(* Logix 5000 project; controller QW361 vendor 1 type 14 code 107 rev 32.11; software revision 32.00; part 20 of 20 *)
(* tags used below, declared in another part *)
   DG1 : MOTOR;   // Diesel generator
   FIT001 : PRANALOG;   // Station discharge flow
   FIT001_CA : ALM;   // Station discharge flow calibrate mode alarm
   FIT001_FL : ALM;   // Station discharge flow sensor fail alarm
   FIT001_hh : ALM;   // Station discharge flow high high alarm
   FIT001_hi : ALM;   // Station discharge flow high alarm
   FIT001_ll : ALM;   // Station discharge flow low low alarm
   FIT001_lo : ALM;   // Station discharge flow low alarm
   FunctionBlock_Cycle_Time : REAL;   // Main Task Cycle Time in mseconds
   LIT001 : PRANALOG;   // Wet well level
   LIT001_CA : ALM;   // Wet well level calibrate mode alarm
   LIT001_FL : ALM;   // Wet well level sensor fail alarm
   LIT001_hh : ALM;   // Wet well level high high alarm
   LIT001_hi : ALM;   // Wet well level high alarm
   LIT001_ll : ALM;   // Wet well level low low alarm
   LIT001_lo : ALM;   // Wet well level low alarm
   P001 : MOTOR;   // Raw sewage pump 1
   P002 : MOTOR;   // Raw sewage pump 2
   pranalog_pwrup_done : BOOL;
   report15_data : LogRecord15[800];
   report15_row_qty : DINT;
   report5_data : LogRecord5[2400];
   report5_row_qty : DINT;
   report_data : LogRecord[200];
   report_pwrup_done : BOOL;
   report_row_qty : DINT;
   sequence_pwrup_done : BOOL;
   valve_pwrup_done : BOOL;
   WALLCLOCK : DateTime;   // Global date / time
   WALLCLOCK_lock : BOOL;

PROGRAM PranalogProgram   (* main routine Pranalogs *)
VAR
   pranalog : PRANALOG := (MaxEU := 20.0, raw := -0.00625, valid := 1, log := 1, hihiraw := 1, hiraw := 1);
   ratio : REAL;
END_VAR

ROUTINE PranalogRoutine   (* structured text *)
   SBR(pranalog);
   
   (* Pranalog function block *)
   
   (* Does all processing for process analogs *)
   
   (* Calling parameters: *)
   (*     pranalog : PRANALOG *)
   
   (* Globals used: *)
   (*     functionblocktask_cycle_time *)
   
   (* Globals changed: *)
   
   (*-------------------------------------------------------------------------------------------------------------------------------------------------*)
   
   
   (* handle the processed analogs *)
   
   (* if not in calibrate mode and not hold and pranalog.calc is not NAN, set the output to calc, smoothed by lag *)
   IF NOT pranalog.calib AND NOT pranalog.hold AND (pranalog.calc = pranalog.calc) THEN
       IF pranalog.lag = 0.0 THEN
           ratio := 0.0;
       ELSE
           ratio := 2.71828 ** ( 0.0 - FunctionBlock_Cycle_Time / 60000.0 / pranalog.lag );
       END_IF;
   
       pranalog.value := ( ( pranalog.value * ratio ) + ( pranalog.calc * ( 1.0 - ratio ) ) );
   
   	(* Check for NAN and if so, set to .calc *)
   	(*IF (S:V) Then
   		pranalog.value := pranalog.calc;
   	END_IF;*)
   
   END_IF;
   
   (* create conditions for high and low alarms *)
   IF pranalog.value > pranalog.hilim  THEN
       pranalog.hiraw := 1;
   END_IF;
   
   IF pranalog.value > pranalog.hihilim  THEN
       pranalog.hihiraw := 1;
   END_IF;
   
   
   IF pranalog.value < ( pranalog.hilim - pranalog.almdb ) THEN
       pranalog.hiraw := 0;
   END_IF;
   
   IF pranalog.value < ( pranalog.hihilim - pranalog.almdb ) THEN
       pranalog.hihiraw := 0;
   END_IF;
   
   IF pranalog.value < pranalog.lolim THEN
       pranalog.loraw := 1;
   END_IF;
   
   IF pranalog.value < pranalog.lololim THEN
       pranalog.loloraw := 1;
   END_IF;
   
   IF pranalog.value > ( pranalog.lolim + pranalog.almdb ) THEN
       pranalog.loraw := 0;
   END_IF;
   
   IF pranalog.value > ( pranalog.lololim + pranalog.almdb ) THEN
       pranalog.loloraw := 0;
   END_IF;
   
   ret(pranalog);
   
END_ROUTINE

ROUTINE Pranalogs   (* structured text *)
   (* Pranalog processing program *)
   
   (* Does all basic processing for all process analogs by setting up inputs then calling the pranalog function block for each *)
   
   (* Globals used: *)
   
   (* Globals changed: *)
   (*     pranalog_pwrup_done *)
   (*     pwrup_dlayd *)
   (*     cycle_time *)
   (*     each motor *)
   
   (*-------------------------------------------------------------------------------------------------------------------------------------------------*)
   
   
   
   (* process each process analog as follows: (note these comments are only shown here for brevity) *)
   (*     1. set up inputs (specific to each analog and commented *)
   (*     2. call the pranalog processing function block *)
   
   
   (************ insert pranalogs here ***************)
   
   
   
   
   (* LIT001 Wet well level *)
   
   (* set up the inputs *)
   LIT001.raw := LIT001.raw;
   LIT001.hold := 0;
   LIT001.valid := NOT ( LIT001.raw < -2.5 OR LIT001.raw > 102.5 ); //Standard
   //Standard
   IF LIT001.raw < 0 THEN
       LIT001.calc := LIT001.MinEU;
   ELSE
       LIT001.calc := LIT001.raw / 100.0 * (LIT001.MaxEU - LIT001.MinEU) + LIT001.MinEU;
   END_IF;
   LIT001.log := 1;
   
   (* process the analog *)
   JSR( PranalogRoutine, 1, LIT001, LIT001 );
   LIT001_hi.raw := LIT001.hiraw;
   LIT001_lo.raw := LIT001.loraw;
   LIT001_hh.raw := LIT001.hihiraw;
   LIT001_ll.raw := LIT001.loloraw;
   LIT001_CA.raw := LIT001.calib;
   LIT001_FL.raw := NOT LIT001.valid;
   
   
   (* FIT001 Station discharge flow *)
   
   (* set up the inputs *)
   FIT001.raw := FIT001.raw;
   FIT001.hold := 0;
   FIT001.valid := NOT ( FIT001.raw < -2.5 OR FIT001.raw > 102.5 ); //Standard
   //> 2 % of span
   IF FIT001.raw < 0 THEN
       FIT001.calc := FIT001.MinEU;
   ELSE
       FIT001.calc := FIT001.raw / 100.0 * (FIT001.MaxEU - FIT001.MinEU) + FIT001.MinEU;
   END_IF;
   FIT001.log := 1;
   
   (* process the analog *)
   JSR( PranalogRoutine, 1, FIT001, FIT001 );
   FIT001_hi.raw := FIT001.hiraw;
   FIT001_lo.raw := FIT001.loraw;
   FIT001_hh.raw := FIT001.hihiraw;
   FIT001_ll.raw := FIT001.loloraw;
   FIT001_CA.raw := FIT001.calib;
   FIT001_FL.raw := NOT FIT001.valid;
   
   
   
   
   (* flag that powerup is done *)
   pranalog_pwrup_done := 1;
   
END_ROUTINE
END_PROGRAM

PROGRAM Report15Calcs   (* main routine Reports *)
VAR
   date_time_current : DateTime := (Year := 2022, Month := 5, Day := 3, Hour := 16, Minute := 29, Second := 58, Microsecond := 621793, DayOfWeek := 2, DST_ON := 1);
   date_time_previous : DateTime := (Year := 2022, Month := 5, Day := 3, Hour := 16, Minute := 29, Second := 58, Microsecond := 621793, DayOfWeek := 2, DST_ON := 1);
   DeleteLog : BOOL;   // Switched on by program to delete logs. Resets when delete is complete
   enable_calc : BOOL := 1;
   ForceDelete : BOOL;   // Switch on to delete contents of log
   max_report_tags : DINT := 5;
   max_tag_idx : DINT := 25;
   MinuteCrt : DINT := 29;
   period_end : BOOL;
   report_row : DINT := 284;
   report_tag_qty : DINT := 5;
   run_val : BOOL;
   tag_idx : DINT := 5;
   tag_valid : BOOL := 1;
   tag_value : REAL := 1.0;
END_VAR

ROUTINE LogCalcRoutine   (* structured text *)
   SBR(tag_value, tag_valid, enable_calc, tag_idx);
   
   (* LogCalc Routine *)
   
   (* Does all processing for log calculations *)
   
   (* Calling parameters: *)
   (*	   tag_value : REAL value of the tag *)
   (*	   tag_valid : BOOL validity of information *)
   (*	   tag_idx : SINT tag index *)
   
   (* Globals used: *)
   
   (* Globals changed: *)
   
   (*-------------------------------------------------------------------------------------------------------------------------------------------------*)
   
   (* check value for quality *)
   tag_value := tag_value;
   (*IF (S:V) THEN
   	tag_value := 0;
   	tag_valid := 0;
   	enable_calc := 0;
   END_IF;*)
   
   
   (* only calculate if it is enabled *)
   IF enable_calc THEN
   	(* check for valid data *)
   	IF  NOT (tag_value = tag_value) THEN
   		tag_valid := 0;
   		tag_value := 0;
   	END_IF;
   
   	(* calculate the max and min *)
   
   	(* if this is the first time this hour, set max and min to current value *)
   	IF report15_data[report_row].log_data[tag_idx].time = 0 THEN
   		report15_data[report_row].log_data[tag_idx].max := tag_value;
   		report15_data[report_row].log_data[tag_idx].min := tag_value;
   		report15_data[report_row].log_data[tag_idx].maxminute := MinuteCrt;
   		report15_data[report_row].log_data[tag_idx].minminute := MinuteCrt;
   
   	(* otherwise, check to see if max or min has been exceeded *)
   	ELSE
   		IF tag_value > report15_data[report_row].log_data[tag_idx].max THEN
   		    report15_data[report_row].log_data[tag_idx].max := tag_value;
   			report15_data[report_row].log_data[tag_idx].maxminute := MinuteCrt;
   		ELSIF tag_value < report15_data[report_row].log_data[tag_idx].min THEN
   		    report15_data[report_row].log_data[tag_idx].min := tag_value;
   			report15_data[report_row].log_data[tag_idx].minminute := MinuteCrt;
   		END_IF;
   	END_IF;
   
   
   	(* add to the total *)
   	report15_data[report_row].log_data[tag_idx].total := report15_data[report_row].log_data[tag_idx].total + FunctionBlock_Cycle_Time / 1000 * tag_value;
   
   	(* add to the time *)
   	report15_data[report_row].log_data[tag_idx].time := report15_data[report_row].log_data[tag_idx].time + FunctionBlock_Cycle_Time / 1000;
   
   	(* Valid *)
   	IF NOT (tag_valid) THEN
   		report15_data[report_row].log_data[tag_idx].valid := 0;
   	END_IF;
   
   END_IF;
END_ROUTINE

ROUTINE LogDeleteRoutine   (* structured text *)
// Deletes log and resets it to Zero
   SBR();
   
   (* LogDelete Routine *)
   
   (* Does all processing to clear out Log *)
   
   (* Calling parameters: *)
   
   (* Globals used: *)
   
   (* Globals changed: *)
   
   (*-------------------------------------------------------------------------------------------------------------------------------------------------*)
   
   
   (* set the timestamp for the finished row *)
   report15_data[report_row].time.Year := 0;
   report15_data[report_row].time.Month := 0;
   report15_data[report_row].time.Day := 0;
   report15_data[report_row].time.Hour := 0;
   report15_data[report_row].time.Minute := 0;
   report15_data[report_row].time.Second := 0;
   report15_data[report_row].time.DST_ON := 0;
   
   (* Go to next record *)
   report_row := report_row + 1;
   IF report_row >= report15_row_qty THEN
   	report_row := 0;
   END_IF;
   
   (* clear the timestamp for the new row *)
   report15_data[report_row].time.Year := 0;
   report15_data[report_row].time.Month := 0;
   report15_data[report_row].time.Day := 0;
   report15_data[report_row].time.Hour := 0;
   report15_data[report_row].time.Minute := 0;
   report15_data[report_row].time.Second := 0;
   report15_data[report_row].time.DST_ON := 0;
   
   (* Do initialisation for the new record *)
   FOR tag_idx := 0 to report_tag_qty - 1 DO
   	report15_data[report_row].log_data[tag_idx].min := 0;
   	report15_data[report_row].log_data[tag_idx].max := 0;
   	report15_data[report_row].log_data[tag_idx].total := 0;
   	report15_data[report_row].log_data[tag_idx].time := 0;
   	report15_data[report_row].log_data[tag_idx].valid := 1;
   END_FOR;
   
   (* Do initialisation for the new record *)
   SIZE(report15_data[report_row].log_data[0],0,max_report_tags);
   max_report_tags := report_tag_qty;  // to be deleted if above line is correct  this will allow clearing of the full table
   FOR tag_idx := 0 to max_report_tags - 1 DO
   	report15_data[report_row].log_data[tag_idx].min := 0;
   	report15_data[report_row].log_data[tag_idx].max := 0;
   	report15_data[report_row].log_data[tag_idx].total := 0;
   	report15_data[report_row].log_data[tag_idx].time := 0;
   	report15_data[report_row].log_data[tag_idx].minminute := 0;
   	report15_data[report_row].log_data[tag_idx].maxminute := 0;
   	report15_data[report_row].log_data[tag_idx].valid := 1;
   END_FOR;
   
   (* If this is the last row to delete (i.e. row 0) end the delete *)
   IF report_row = 0 THEN
   	DeleteLog := 0;
   END_IF;
END_ROUTINE

ROUTINE LogMotorRoutine   (* structured text *)
   SBR(run_val, tag_idx);
   
   IF run_val THEN
   	JSR(LogCalcRoutine, 4 , 1.0, 1, 1, tag_idx);
   ELSE
   	JSR(LogCalcRoutine, 4 , 0.0, 1, 1, tag_idx);
   END_IF;
   
END_ROUTINE

ROUTINE LogSaveRoutine   (* structured text *)
   SBR();
   
   (* LogSave Routine *)
   
   (* Does all processing for saving log data at the end of the hour *)
   
   (* Calling parameters: *)
   
   (* Globals used: *)
   
   (* Globals changed: *)
   
   (*-------------------------------------------------------------------------------------------------------------------------------------------------*)
   
   
   (* set the timestamp for the finished row *)
   report15_data[report_row].time.Year := date_time_previous.Year;
   report15_data[report_row].time.Month := date_time_previous.Month;
   report15_data[report_row].time.Day := date_time_previous.Day;
   report15_data[report_row].time.Hour := date_time_previous.Hour;
   report15_data[report_row].time.Minute := date_time_previous.Minute;
   report15_data[report_row].time.Second := date_time_previous.Second;
   report15_data[report_row].time.DST_ON := date_time_previous.DST_ON;
   
   (* Go to next record *)
   report_row := report_row + 1;
   IF report_row >= report15_row_qty THEN
   	report_row := 0;
   END_IF;
   
   (* clear the timestamp for the new row *)
   report15_data[report_row].time.Year := 0;
   report15_data[report_row].time.Month := 0;
   report15_data[report_row].time.Day := 0;
   report15_data[report_row].time.Hour := 0;
   report15_data[report_row].time.Minute := 0;
   report15_data[report_row].time.Second := 0;
   report15_data[report_row].time.DST_ON := 0;
   
   (* Do initialisation for the new record *)
   FOR tag_idx := 0 to report_tag_qty - 1 DO
   	report15_data[report_row].log_data[tag_idx].min := 0;
   	report15_data[report_row].log_data[tag_idx].max := 0;
   	report15_data[report_row].log_data[tag_idx].total := 0;
   	report15_data[report_row].log_data[tag_idx].time := 0;
   	report15_data[report_row].log_data[tag_idx].valid := 1;
   END_FOR;
   
   (* Do initialisation for the new record *)
   SIZE(report15_data[report_row].log_data[0],0,max_report_tags);
   max_report_tags := report_tag_qty;  // to be deleted if above line is correct  this will allow clearing of the full table
   FOR tag_idx := 0 to max_report_tags - 1 DO
   	report15_data[report_row].log_data[tag_idx].min := 0;
   	report15_data[report_row].log_data[tag_idx].max := 0;
   	report15_data[report_row].log_data[tag_idx].total := 0;
   	report15_data[report_row].log_data[tag_idx].time := 0;
   	report15_data[report_row].log_data[tag_idx].minminute := 0;
   	report15_data[report_row].log_data[tag_idx].maxminute := 0;
   	report15_data[report_row].log_data[tag_idx].valid := 1;
   END_FOR;
END_ROUTINE

ROUTINE Reports   (* structured text *)
   (* Report logging processing program *)
   
   (* Does all processing for logging of report data *)
   
   (* Globals used: *)
   
   (* Globals changed: *)
   
   (*-------------------------------------------------------------------------------------------------------------------------------------------------*)
   
   
   //**********************to be adjusted by programmer ********************************
   SIZE(report15_data[0],0,report15_row_qty);
   SIZE(report15_data[0].log_data[0],0,report_tag_qty);
   //***********************************************************************************
   
   (* Get current date/time *)
   IF NOT WALLCLOCK_lock THEN
   	cop( WALLCLOCK, date_time_current, 1);
   END_IF;
   
   (* adjust previous hour if dst changed *)
   IF date_time_current.DST_ON AND NOT date_time_previous.DST_ON THEN
   	date_time_previous.Hour := date_time_previous.Hour + 1;
   ELSIF NOT date_time_current.DST_ON AND date_time_previous.DST_ON THEN
   	date_time_previous.Hour := date_time_previous.Hour - 1;
   END_IF;
   
   (* Detect 15 minute change to see if the period is over *)
   IF date_time_current.Minute <> date_time_previous.Minute THEN
   	period_end := (date_time_current.Minute / 15) <> (date_time_previous.Minute / 15);
   ELSE
   	period_end := 0;
   END_IF;
   
   (* if the hour just ended, save the new hour's data *)
   IF period_end THEN
   	JSR(LogSaveRoutine);
   END_IF;
   
   (* delete log logic, used to clear out data log *)
   If ForceDelete AND NOT DeleteLog THEN
   	DeleteLog := 1;
   	report_row := 1;
   END_IF;
   If DeleteLog THEN
   	JSR(LogDeleteRoutine);
   END_IF;
   ForceDelete := 0;
   
   
   MinuteCrt := date_time_current.Minute;
   
   
   (************ insert logs here ***************)
   
   
   (* keep track of the last date for the end of the hour *)
   COP(date_time_current,date_time_previous,1);
   
END_ROUTINE
END_PROGRAM

PROGRAM Report5Calcs   (* main routine Reports *)
VAR
   date_time_current : DateTime := (Year := 2022, Month := 5, Day := 3, Hour := 16, Minute := 29, Second := 58, Microsecond := 621793, DayOfWeek := 2, DST_ON := 1);
   date_time_previous : DateTime := (Year := 2022, Month := 5, Day := 3, Hour := 16, Minute := 29, Second := 58, Microsecond := 621793, DayOfWeek := 2, DST_ON := 1);
   DeleteLog : BOOL;   // Switched on by program to delete logs. Resets when delete is complete
   enable_calc : BOOL := 1;
   ForceDelete : BOOL;   // Switch on to delete contents of log
   max_report_tags : DINT := 5;
   max_tag_idx : DINT := 25;
   MinuteCrt : DINT := 29;
   period_end : BOOL;
   report_row : DINT := 419;
   report_tag_qty : DINT := 5;
   run_val : BOOL;
   tag_idx : DINT;
   tag_valid : BOOL := 1;
   tag_value : REAL := 1.0;
END_VAR

ROUTINE LogCalcRoutine   (* structured text *)
   SBR(tag_value, tag_valid, enable_calc, tag_idx);
   
   (* LogCalc Routine *)
   
   (* Does all processing for log calculations *)
   
   (* Calling parameters: *)
   (*	   tag_value : REAL value of the tag *)
   (*	   tag_valid : BOOL validity of information *)
   (*	   tag_idx : SINT tag index *)
   
   (* Globals used: *)
   
   (* Globals changed: *)
   
   (*-------------------------------------------------------------------------------------------------------------------------------------------------*)
   
   (* check value for quality *)
   tag_value := tag_value;
   (*IF (S:V) THEN
   	tag_value := 0;
   	tag_valid := 0;
   	enable_calc := 0;
   END_IF; *)
   
   
   (* only calculate if it is enabled *)
   IF enable_calc THEN
   	(* check for valid data *)
   	IF  NOT (tag_value = tag_value) THEN
   		tag_valid := 0;
   		tag_value := 0;
   	END_IF;
   
   	(* calculate the max and min *)
   
   	(* if this is the first time this hour, set max and min to current value *)
   	IF report5_data[report_row].log_data[tag_idx].time = 0 THEN
   		report5_data[report_row].log_data[tag_idx].max := tag_value;
   		report5_data[report_row].log_data[tag_idx].min := tag_value;
   		report5_data[report_row].log_data[tag_idx].maxminute := MinuteCrt;
   		report5_data[report_row].log_data[tag_idx].minminute := MinuteCrt;
   
   	(* otherwise, check to see if max or min has been exceeded *)
   	ELSE
   		IF tag_value > report5_data[report_row].log_data[tag_idx].max THEN
   		    report5_data[report_row].log_data[tag_idx].max := tag_value;
   			report5_data[report_row].log_data[tag_idx].maxminute := MinuteCrt;
   		ELSIF tag_value < report5_data[report_row].log_data[tag_idx].min THEN
   		    report5_data[report_row].log_data[tag_idx].min := tag_value;
   			report5_data[report_row].log_data[tag_idx].minminute := MinuteCrt;
   		END_IF;
   	END_IF;
   
   
   	(* add to the total *)
   	report5_data[report_row].log_data[tag_idx].total := report5_data[report_row].log_data[tag_idx].total + FunctionBlock_Cycle_Time / 1000 * tag_value;
   
   	(* add to the time *)
   	report5_data[report_row].log_data[tag_idx].time := report5_data[report_row].log_data[tag_idx].time + FunctionBlock_Cycle_Time / 1000;
   
   	(* Valid *)
   	IF NOT (tag_valid) THEN
   		report5_data[report_row].log_data[tag_idx].valid := 0;
   	END_IF;
   
   END_IF;
END_ROUTINE

ROUTINE LogDeleteRoutine   (* structured text *)
// Deletes log and resets it to Zero
   SBR();
   
   (* LogDelete Routine *)
   
   (* Does all processing to clear out Log *)
   
   (* Calling parameters: *)
   
   (* Globals used: *)
   
   (* Globals changed: *)
   
   (*-------------------------------------------------------------------------------------------------------------------------------------------------*)
   
   
   (* set the timestamp for the finished row *)
   report5_data[report_row].time.Year := 0;
   report5_data[report_row].time.Month := 0;
   report5_data[report_row].time.Day := 0;
   report5_data[report_row].time.Hour := 0;
   report5_data[report_row].time.Minute := 0;
   report5_data[report_row].time.Second := 0;
   report5_data[report_row].time.DST_ON := 0;
   
   (* Go to next record *)
   report_row := report_row + 1;
   IF report_row >= report5_row_qty THEN
   	report_row := 0;
   END_IF;
   
   (* clear the timestamp for the new row *)
   report5_data[report_row].time.Year := 0;
   report5_data[report_row].time.Month := 0;
   report5_data[report_row].time.Day := 0;
   report5_data[report_row].time.Hour := 0;
   report5_data[report_row].time.Minute := 0;
   report5_data[report_row].time.Second := 0;
   report5_data[report_row].time.DST_ON := 0;
   
   (* Do initialisation for the new record *)
   FOR tag_idx := 0 to report_tag_qty - 1 DO
   	report5_data[report_row].log_data[tag_idx].min := 0;
   	report5_data[report_row].log_data[tag_idx].max := 0;
   	report5_data[report_row].log_data[tag_idx].total := 0;
   	report5_data[report_row].log_data[tag_idx].time := 0;
   	report5_data[report_row].log_data[tag_idx].valid := 1;
   END_FOR;
   
   (* Do initialisation for the new record *)
   SIZE(report5_data[report_row].log_data[0],0,max_report_tags);
   max_report_tags := report_tag_qty;  // to be deleted if above line is correct  this will allow clearing of the full table
   FOR tag_idx := 0 to max_report_tags - 1 DO
   	report5_data[report_row].log_data[tag_idx].min := 0;
   	report5_data[report_row].log_data[tag_idx].max := 0;
   	report5_data[report_row].log_data[tag_idx].total := 0;
   	report5_data[report_row].log_data[tag_idx].time := 0;
   	report5_data[report_row].log_data[tag_idx].minminute := 0;
   	report5_data[report_row].log_data[tag_idx].maxminute := 0;
   	report5_data[report_row].log_data[tag_idx].valid := 1;
   END_FOR;
   
   (* If this is the last row to delete (i.e. row 0) end the delete *)
   IF report_row = 0 THEN
   	DeleteLog := 0;
   END_IF;
END_ROUTINE

ROUTINE LogMotorRoutine   (* structured text *)
   SBR(run_val, tag_idx);
   
   IF run_val THEN
   	JSR(LogCalcRoutine, 4 , 1.0, 1, 1, tag_idx);
   ELSE
   	JSR(LogCalcRoutine, 4 , 0.0, 1, 1, tag_idx);
   END_IF;
   
END_ROUTINE

ROUTINE LogSaveRoutine   (* structured text *)
   SBR();
   
   (* LogSave Routine *)
   
   (* Does all processing for saving log data at the end of the hour *)
   
   (* Calling parameters: *)
   
   (* Globals used: *)
   
   (* Globals changed: *)
   
   (*-------------------------------------------------------------------------------------------------------------------------------------------------*)
   
   
   (* set the timestamp for the finished row *)
   report5_data[report_row].time.Year := date_time_previous.Year;
   report5_data[report_row].time.Month := date_time_previous.Month;
   report5_data[report_row].time.Day := date_time_previous.Day;
   report5_data[report_row].time.Hour := date_time_previous.Hour;
   report5_data[report_row].time.Minute := date_time_previous.Minute;
   report5_data[report_row].time.Second := date_time_previous.Second;
   report5_data[report_row].time.DST_ON := date_time_previous.DST_ON;
   
   (* Go to next record *)
   report_row := report_row + 1;
   IF report_row >= report5_row_qty THEN
   	report_row := 0;
   END_IF;
   
   (* clear the timestamp for the new row *)
   report5_data[report_row].time.Year := 0;
   report5_data[report_row].time.Month := 0;
   report5_data[report_row].time.Day := 0;
   report5_data[report_row].time.Hour := 0;
   report5_data[report_row].time.Minute := 0;
   report5_data[report_row].time.Second := 0;
   report5_data[report_row].time.DST_ON := 0;
   
   (* Do initialisation for the new record *)
   FOR tag_idx := 0 to report_tag_qty - 1 DO
   	report5_data[report_row].log_data[tag_idx].min := 0;
   	report5_data[report_row].log_data[tag_idx].max := 0;
   	report5_data[report_row].log_data[tag_idx].total := 0;
   	report5_data[report_row].log_data[tag_idx].time := 0;
   	report5_data[report_row].log_data[tag_idx].valid := 1;
   END_FOR;
   
   (* Do initialisation for the new record *)
   SIZE(report5_data[report_row].log_data[0],0,max_report_tags);
   max_report_tags := report_tag_qty;  // to be deleted if above line is correct  this will allow clearing of the full table
   FOR tag_idx := 0 to max_report_tags - 1 DO
   	report5_data[report_row].log_data[tag_idx].min := 0;
   	report5_data[report_row].log_data[tag_idx].max := 0;
   	report5_data[report_row].log_data[tag_idx].total := 0;
   	report5_data[report_row].log_data[tag_idx].time := 0;
   	report5_data[report_row].log_data[tag_idx].minminute := 0;
   	report5_data[report_row].log_data[tag_idx].maxminute := 0;
   	report5_data[report_row].log_data[tag_idx].valid := 1;
   END_FOR;
END_ROUTINE

ROUTINE Reports   (* structured text *)
   (* Report logging processing program *)
   
   (* Does all processing for logging of report data *)
   
   (* Globals used: *)
   
   (* Globals changed: *)
   
   (*-------------------------------------------------------------------------------------------------------------------------------------------------*)
   
   
   //**********************to be adjusted by programmer ********************************
   SIZE(report5_data[0],0,report5_row_qty);
   SIZE(report5_data[0].log_data[0],0,report_tag_qty);
   //***********************************************************************************
   
   (* Get current date/time *)
   IF NOT WALLCLOCK_lock THEN
   	cop( WALLCLOCK, date_time_current, 1);
   END_IF;
   
   (* adjust previous hour if dst changed *)
   IF date_time_current.DST_ON AND NOT date_time_previous.DST_ON THEN
   	date_time_previous.Hour := date_time_previous.Hour + 1;
   ELSIF NOT date_time_current.DST_ON AND date_time_previous.DST_ON THEN
   	date_time_previous.Hour := date_time_previous.Hour - 1;
   END_IF;
   
   (* Detect 5 minute change to see if the period is over *)
   IF date_time_current.Minute <> date_time_previous.Minute THEN
   	period_end := (date_time_current.Minute / 5) <> (date_time_previous.Minute / 5);
   ELSE
   	period_end := 0;
   END_IF;
   
   (* if the hour just ended, save the new hour's data *)
   IF period_end THEN
   	JSR(LogSaveRoutine);
   END_IF;
   
   (* delete log logic, used to clear out data log *)
   If ForceDelete AND NOT DeleteLog THEN
   	DeleteLog := 1;
   	report_row := 1;
   END_IF;
   If DeleteLog THEN
   	JSR(LogDeleteRoutine);
   END_IF;
   ForceDelete := 0;
   
   MinuteCrt := date_time_current.Minute;
   
   
   (************ insert logs here ***************)
   
   
   JSR( LogCalcRoutine, 4, 1.0, 1, 1, 0);  //duration
   
   
   (* keep track of the last date for the end of the hour *)
   COP(date_time_current,date_time_previous,1);
   
END_ROUTINE
END_PROGRAM

PROGRAM ReportCalcs   (* main routine Reports *)
VAR
   date_time_current : DateTime := (Year := 2022, Month := 5, Day := 3, Hour := 16, Minute := 29, Second := 58, Microsecond := 621793, DayOfWeek := 2, DST_ON := 1);
   date_time_previous : DateTime := (Year := 2022, Month := 5, Day := 3, Hour := 16, Minute := 29, Second := 58, Microsecond := 621793, DayOfWeek := 2, DST_ON := 1);
   DeleteLog : BOOL;   // Switched on by program to delete logs. Resets when delete is complete
   enable_calc : BOOL := 1;
   ForceDelete : BOOL;   // Switch on to delete contents of log
   hour_end : BOOL;
   max_report_tags : DINT := 20;
   max_tag_idx : DINT := 25;
   MinuteCrt : DINT := 29;
   report_row : DINT := 167;
   run_val : BOOL;
   tag_idx : DINT := 5;
   tag_valid : BOOL := 1;
   tag_value : REAL;
END_VAR

ROUTINE LogCalcRoutine   (* structured text *)
   SBR(tag_value, tag_valid, enable_calc, tag_idx);
   
   (* LogCalc Routine *)
   
   (* Does all processing for log calculations *)
   
   (* Calling parameters: *)
   (*	   tag_value : REAL value of the tag *)
   (*	   tag_valid : BOOL validity of information *)
   (*	   tag_idx : SINT tag index *)
   
   (* Globals used: *)
   
   (* Globals changed: *)
   
   (*-------------------------------------------------------------------------------------------------------------------------------------------------*)
   
   (* check value for quality *)
   tag_value := tag_value;
   (*IF (S:V) THEN
   	tag_value := 0;
   	tag_valid := 0;
   	enable_calc := 0;
   END_IF;*)
   
   (* only calculate if it is enabled *)
   IF enable_calc THEN
   	(* check for valid data *)
   	IF  NOT (tag_value = tag_value) THEN
   		tag_valid := 0;
   		tag_value := 0;
   	END_IF;
   
   	(* calculate the max and min *)
   
   	(* if this is the first time this hour, set max and min to current value *)
   	IF report_data[report_row].log_data[tag_idx].time = 0 THEN
   		report_data[report_row].log_data[tag_idx].max := tag_value;
   		report_data[report_row].log_data[tag_idx].min := tag_value;
   		report_data[report_row].log_data[tag_idx].maxminute := MinuteCrt;
   		report_data[report_row].log_data[tag_idx].minminute := MinuteCrt;
   
   	(* otherwise, check to see if max or min has been exceeded *)
   	ELSE
   		IF tag_value > report_data[report_row].log_data[tag_idx].max THEN
   		    report_data[report_row].log_data[tag_idx].max := tag_value;
   			report_data[report_row].log_data[tag_idx].maxminute := MinuteCrt;
   		ELSIF tag_value < report_data[report_row].log_data[tag_idx].min THEN
   		    report_data[report_row].log_data[tag_idx].min := tag_value;
   			report_data[report_row].log_data[tag_idx].minminute := MinuteCrt;
   		END_IF;
   	END_IF;
   
   
   	(* add to the total *)
   	report_data[report_row].log_data[tag_idx].total := report_data[report_row].log_data[tag_idx].total + FunctionBlock_Cycle_Time / 1000 * tag_value;
   
   	(* add to the time *)
   	report_data[report_row].log_data[tag_idx].time := report_data[report_row].log_data[tag_idx].time + FunctionBlock_Cycle_Time / 1000;
   
   	(* Valid *)
   	IF NOT (tag_valid) THEN
   		report_data[report_row].log_data[tag_idx].valid := 0;
   	END_IF;
   
   END_IF;
END_ROUTINE

ROUTINE LogDeleteRoutine   (* structured text *)
// Deletes log and resets it to Zero
   SBR();
   
   (* LogDelete Routine *)
   
   (* Does all processing to clear out Log *)
   
   (* Calling parameters: *)
   
   (* Globals used: *)
   
   (* Globals changed: *)
   
   (*-------------------------------------------------------------------------------------------------------------------------------------------------*)
   
   
   (* set the timestamp for the finished row *)
   report_data[report_row].time.Year := 0;
   report_data[report_row].time.Month := 0;
   report_data[report_row].time.Day := 0;
   report_data[report_row].time.Hour := 0;
   report_data[report_row].time.Minute := 0;
   report_data[report_row].time.Second := 0;
   report_data[report_row].time.DST_ON := 0;
   
   (* Go to next record *)
   report_row := report_row + 1;
   IF report_row >= report_row_qty THEN
   	report_row := 0;
   END_IF;
   
   (* clear the timestamp for the new row *)
   report_data[report_row].time.Year := 0;
   report_data[report_row].time.Month := 0;
   report_data[report_row].time.Day := 0;
   report_data[report_row].time.Hour := 0;
   report_data[report_row].time.Minute := 0;
   report_data[report_row].time.Second := 0;
   report_data[report_row].time.DST_ON := 0;
   
   (* Do initialisation for the new record *)
   FOR tag_idx := 0 to report_tag_qty - 1 DO
   	report_data[report_row].log_data[tag_idx].min := 0;
   	report_data[report_row].log_data[tag_idx].max := 0;
   	report_data[report_row].log_data[tag_idx].total := 0;
   	report_data[report_row].log_data[tag_idx].time := 0;
   	report_data[report_row].log_data[tag_idx].valid := 1;
   END_FOR;
   
   (* Do initialisation for the new record *)
   SIZE(report_data[report_row].log_data[0],0,max_report_tags);
   max_report_tags := report_tag_qty;  // to be deleted if above line is correct  this will allow clearing of the full table
   FOR tag_idx := 0 to max_report_tags - 1 DO
   	report_data[report_row].log_data[tag_idx].min := 0;
   	report_data[report_row].log_data[tag_idx].max := 0;
   	report_data[report_row].log_data[tag_idx].total := 0;
   	report_data[report_row].log_data[tag_idx].time := 0;
   	report_data[report_row].log_data[tag_idx].minminute := 0;
   	report_data[report_row].log_data[tag_idx].maxminute := 0;
   	report_data[report_row].log_data[tag_idx].valid := 1;
   END_FOR;
   
   (* If this is the last row to delete (i.e. row 0) end the delete *)
   IF report_row = 0 THEN
   	DeleteLog := 0;
   END_IF;
END_ROUTINE

ROUTINE LogMotorRoutine   (* structured text *)
   SBR(run_val, tag_idx);
   
   IF run_val THEN
   	JSR(LogCalcRoutine, 4 , 1.0, 1, 1, tag_idx);
   ELSE
   	JSR(LogCalcRoutine, 4 , 0.0, 1, 1, tag_idx);
   END_IF;
   
END_ROUTINE

ROUTINE LogSaveRoutine   (* structured text *)
   SBR();
   
   (* LogSave Routine *)
   
   (* Does all processing for saving log data at the end of the hour *)
   
   (* Calling parameters: *)
   
   (* Globals used: *)
   
   (* Globals changed: *)
   
   (*-------------------------------------------------------------------------------------------------------------------------------------------------*)
   
   
   (* set the timestamp for the finished row *)
   report_data[report_row].time.Year := date_time_previous.Year;
   report_data[report_row].time.Month := date_time_previous.Month;
   report_data[report_row].time.Day := date_time_previous.Day;
   report_data[report_row].time.Hour := date_time_previous.Hour;
   report_data[report_row].time.Minute := date_time_previous.Minute;
   report_data[report_row].time.Second := date_time_previous.Second;
   report_data[report_row].time.DST_ON := date_time_previous.DST_ON;
   
   (* Go to next record *)
   report_row := report_row + 1;
   IF report_row >= report_row_qty THEN
   	report_row := 0;
   END_IF;
   
   (* clear the timestamp for the new row *)
   report_data[report_row].time.Year := 0;
   report_data[report_row].time.Month := 0;
   report_data[report_row].time.Day := 0;
   report_data[report_row].time.Hour := 0;
   report_data[report_row].time.Minute := 0;
   report_data[report_row].time.Second := 0;
   report_data[report_row].time.DST_ON := 0;
   
   (* Do initialisation for the new record *)
   FOR tag_idx := 0 to report_tag_qty - 1 DO
   	report_data[report_row].log_data[tag_idx].min := 0;
   	report_data[report_row].log_data[tag_idx].max := 0;
   	report_data[report_row].log_data[tag_idx].total := 0;
   	report_data[report_row].log_data[tag_idx].time := 0;
   	report_data[report_row].log_data[tag_idx].valid := 1;
   END_FOR;
   
   (* Do initialisation for the new record *)
   SIZE(report_data[report_row].log_data[0],0,max_report_tags);
   max_report_tags := report_tag_qty;  // to be deleted if above line is correct  this will allow clearing of the full table
   FOR tag_idx := 0 to max_report_tags - 1 DO
   	report_data[report_row].log_data[tag_idx].min := 0;
   	report_data[report_row].log_data[tag_idx].max := 0;
   	report_data[report_row].log_data[tag_idx].total := 0;
   	report_data[report_row].log_data[tag_idx].time := 0;
   	report_data[report_row].log_data[tag_idx].minminute := 0;
   	report_data[report_row].log_data[tag_idx].maxminute := 0;
   	report_data[report_row].log_data[tag_idx].valid := 1;
   END_FOR;
END_ROUTINE

ROUTINE Reports   (* structured text *)
   (* Report logging processing program *)
   
   (* Does all processing for logging of report data *)
   
   (* Globals used: *)
   
   (* Globals changed: *)
   
   (*-------------------------------------------------------------------------------------------------------------------------------------------------*)
   
   
   //**********************to be adjusted by programmer ********************************
   SIZE(report_data[0].log_data[0],0,report_tag_qty);
   SIZE(report_data[0],0,report_row_qty);
   //***********************************************************************************
   
   (* Get current date/time *)
   IF NOT WALLCLOCK_lock THEN
   	cop( WALLCLOCK, date_time_current, 1);
   END_IF;
   
   (* adjust previous hour if dst changed *)
   IF date_time_current.DST_ON AND NOT date_time_previous.DST_ON THEN
   	date_time_previous.Hour := date_time_previous.Hour + 1;
   ELSIF NOT date_time_current.DST_ON AND date_time_previous.DST_ON THEN
   	date_time_previous.Hour := date_time_previous.Hour - 1;
   END_IF;
   
   (* Detect hour change to see if the period is over *)
   IF date_time_current.Hour <> date_time_previous.Hour THEN
   	hour_end := 1;
   ELSE
   	hour_end := 0;
   END_IF;
   
   (* if the hour just ended, save the new hour's data *)
   IF hour_end THEN
   	JSR(LogSaveRoutine);
   END_IF;
   
   (* delete log logic, used to clear out data log *)
   If ForceDelete AND NOT DeleteLog THEN
   	DeleteLog := 1;
   	report_row := 1;
   END_IF;
   If DeleteLog THEN
   	JSR(LogDeleteRoutine);
   END_IF;
   ForceDelete := 0;
   
   
   MinuteCrt := date_time_current.Minute;
   
   JSR( LogCalcRoutine, 4, 1.0, 1, 1, 0);  //duration
   (************ insert logs here ***************)
   
   JSR( LogMotorRoutine, 2, P001.run_sts, 1 );  //P001 - Raw sewage pump 1
   JSR( LogMotorRoutine, 2, P002.run_sts, 2 );  //P002 - Raw sewage pump 2
   JSR( LogMotorRoutine, 2, DG1.run_sts, 3 );  //DG1 - Diesel generator
   JSR( LogCalcRoutine, 4, LIT001.value, LIT001.valid, LIT001.log, 4);  //LIT001 - Wet well level
   JSR( LogCalcRoutine, 4, FIT001.value, FIT001.valid, FIT001.log, 5);  //FIT001 - Station discharge flow
   
   
   (* keep track of the last date for the end of the hour *)
   COP(date_time_current,date_time_previous,1);
   
   (* flag that powerup is done *)
   report_pwrup_done := 1;
   
END_ROUTINE
END_PROGRAM

PROGRAM SequenceProgram   (* main routine Sequences *)
VAR
   sequence : SEQUENCE1 := (auto := 1, abort_to_step := 20, step_no := 14, step_done := 1, advance := 1);
END_VAR

ROUTINE SequenceRoutine   (* structured text *)
   SBR( sequence );
   
   (* Sequence function block *)
   
   (* Does all processing for sequence control *)
   
   (* Calling parameters: *)
   (*     sequence : SEQUENCE *)
   
   (* Globals used: *)
   
   (* Globals changed: *)
   
   (*-------------------------------------------------------------------------------------------------------------------------------------------------*)
   
   
   (* if the sequence is not running, check to see if it should be started *)
   IF NOT sequence.run_sts THEN
   
   	(* start sequence if required *)
   	IF
   			sequence.permit
   		AND
   			(
   				sequence.start_man
   			OR
   				sequence.start_auto
   			)
   	THEN
   
   		(* if we just started, then reset all the parameters *)
   		sequence.run_sts := 1;
   		sequence.abort_step := 0;
   		sequence.step_no := 1;
   		sequence.step_time := 0;
   
   	END_IF;
   
   (* if we are running, check for advance or abort *)
   ELSE
   
   	(* pre-calculate the advance control *)
   	sequence.advance := sequence.auto AND sequence.step_done OR NOT sequence.auto AND sequence.advance_man;
   
   	(* abort if required *)
   	IF (sequence.abort_man OR NOT sequence.permit) AND (sequence.abort_step = 0) THEN
   		sequence.abort_step := sequence.step_no;
   		sequence.step_no := sequence.abort_to_step;
   		sequence.step_time := 0;
   
   	(* advance if required *)
   	ELSIF sequence.advance THEN
   		sequence.step_no := sequence.step_no + 1;
   		sequence.step_time := 0;
   
   	(* no abort or advance, so accumulate step time *)
   	ELSE
   		sequence.step_time := sequence.step_time + (FunctionBlock_Cycle_Time / 1000);
   	END_IF;
   
   END_IF;
   
   (* reset the momentaries *)
   IF sequence.start_man THEN sequence.start_man := 0; END_IF;
   IF sequence.advance_man THEN sequence.advance_man := 0; END_IF;
   IF sequence.abort_man THEN sequence.abort_man := 0; END_IF;
   
   RET( sequence );
   
   
END_ROUTINE

ROUTINE Sequences   (* structured text *)
   (* Main processing program *)
   
   (* Call all Sequence subroutine for equipment *)
   
   (* Globals used: *)
   
   (* Globals changed: *)
   
   
   (************ insert sequences here ***************)
   
   
   (* flag that powerup is done *)
   sequence_pwrup_done := 1;
   
END_ROUTINE
END_PROGRAM

PROGRAM ValveProgram   (* main routine Valves *)
VAR
   fail_pending : BOOL;
   pwrup_dlayd : FBD_TIMER := (TimerEnable := 1, PRE := 2000, ACC := 2000, EN := 1, DN := 1);
   valve : VALVE := (remote := 1, permit := 1, hold_out := 1, close_sts := 1, desired_state := 2, fail_tonr.Reset := 1);
END_VAR

ROUTINE ValveRoutine   (* structured text *)
   SBR(valve);
   
   (* Valve function block *)
   
   (* Does all valve control processing *)
   
   (* Calling parameters: *)
   (*     valve : VALVE *)
   
   (* Globals used: *)
   (*     pwrup_dlayd *)
   
   (* Globals changed: *)
   (*     fail_pending *)
   
   (*-------------------------------------------------------------------------------------------------------------------------------------------------*)
   
   
   (* Load fault time with preset value *)
   valve.fail_tonr.PRE := valve.fail_dlay * 1000;
   valve.fail_tonr.TimerEnable := 1;
   
   
   (* handle the failure logic first *)
   
   (* calculate the fail pending *)
   IF
           NOT valve.remote
       OR
           ( valve.desired_state = 0 AND NOT valve.open_sts AND valve.close_sts )
       OR
           ( valve.desired_state = 1 AND valve.open_sts AND NOT valve.close_sts )
       OR
           valve.desired_state = 2
   	OR
   	    NOT pwrup_dlayd.DN
   THEN
       fail_pending := 0;
   ELSE
       fail_pending := 1;
   END_IF;
   
   (* time the fail pending *)
   valve.fail_tonr.Reset := NOT fail_pending;
   tonr(valve.fail_tonr);
   
   (* calculate the fail and clear if we're not in remote or we just powered up *)
   valve.fail := ( valve.fail AND ( NOT valve.fail_reset AND valve.remote AND pwrup_dlayd.DN ) ) OR valve.fail_tonr.DN;
   
   
   (* handle the valve desired state and outputs *)
   
   (* if we're failed, not remote or not permitted to move or just powered up, set desired state to hold *)
   IF valve.fail OR NOT valve.remote OR NOT valve.permit OR NOT pwrup_dlayd.DN THEN
       valve.desired_state := 2;
   
   (* if not in auto process the manual commands *)
   ELSIF NOT valve.auto THEN
   	IF valve.close_man AND valve.permit THEN
   		valve.desired_state := 0;
   	ELSIF valve.open_man AND valve.permit THEN
   		valve.desired_state := 1;
   	ELSIF valve.hold_man THEN
   		valve.desired_state := 2;
   	END_IF;
   
   (* if in auto process the auto commands*)
   ELSE
   
   	IF valve.close_auto AND valve.permit THEN
   		valve.desired_state := 0;
   	ELSIF valve.open_auto AND valve.permit THEN
   		valve.desired_state := 1;
   	ELSIF valve.hold_auto THEN
   		valve.desired_state := 2;
   	END_IF;
   
   END_IF;
   
   (* create the valve outputs *)
   valve.close_out := valve.desired_state = 0 AND ( valve.open_sts OR NOT valve.close_sts );
   valve.open_out := valve.desired_state = 1 AND ( NOT valve.open_sts OR valve.close_sts );
   valve.hold_out := valve.desired_state = 2;
   valve.runopn_out := valve.desired_state = 1;
   
   
   (* process the momentary resets *)
   
   (* set the momentary resets equal to the current state *)
   IF valve.hold_man THEN valve.hold_man := 0; END_IF;
   IF valve.close_man THEN valve.close_man := 0; END_IF;
   IF valve.open_man THEN valve.open_man := 0; END_IF;
   IF valve.hold_auto THEN valve.hold_auto := 0; END_IF;
   IF valve.close_auto THEN valve.close_auto := 0; END_IF;
   IF valve.open_auto THEN valve.open_auto := 0; END_IF;
   IF valve.fail_reset THEN valve.fail_reset := 0; END_IF;
   
   ret(valve);
   
END_ROUTINE

ROUTINE Valves   (* structured text *)
   (* Valve processing program *)
   
   (* Does all basic processing for all valves by setting up inputs then calling the valve function block for each *)
   
   (* Globals used: *)
   
   (* Globals changed: *)
   (*     valve_pwrup_done *)
   (*     pwrup_dlayd *)
   (*     each valve *)
   
   (*-------------------------------------------------------------------------------------------------------------------------------------------------*)
   
   
   (* use a TONR to delay power recovery *)
   
   pwrup_dlayd.Reset := not valve_pwrup_done;
   TONR(pwrup_dlayd);
   
   
   (* process each valve as follows: (note these comments are only shown here for brevity) *)
   (*     1. set up inputs (specific to each valve and commented *)
   (*     2. call the valve processing function block *)
   (*     3. clear the momentary inputs if they were on *)
   (*     4. get the outputs *)
   
   
   (************ insert valves here ***************)
   
   
   (* flag that powerup is done *)
   valve_pwrup_done := 1;
   
END_ROUTINE
END_PROGRAM
